// TIA Portal V19 export
TYPE "lexchangetray_typeUnEmn_recieve_interface"
// Type: lexchangetray_typeUnEmn_toHandlingXyzRecieve
// Type: lexchangetray_typeUnEmn_toConstraintWorkstationRecieve
// Type: lexchangetray_typeUnEmn_toRollerRecieve
// stored: Access Published
   STRUCT
      roller { S7_SetPoint := 'True'} : "lexchangetray_typeUnEmn_toRollerRecieve";
      constraintWorkstation { S7_SetPoint := 'True'} : "lexchangetray_typeUnEmn_toConstraintWorkstationRecieve";
      handlingXyz { S7_SetPoint := 'True'} : "lexchangetray_typeUnEmn_toHandlingXyzRecieve";
   END_STRUCT;
END_TYPE
